{attribute 'qualified_only'}
{attribute 'strict'}
TYPE E_CONVAYOR_STATE :
(
	uninit,
	idle,
	do_move,
	done,
	pause,
	error
);
END_TYPE

(* stored: Version 1.1.0.1, ProductVersion 3.1.4024.12
   DUT E_CONVAYOR_STATE: Id {a101147d-ea86-4c99-97c2-f80e7395fae2} *)
